SUBAPPLICATION Uebung_080e3 (* Beispiel für E_CTU mit Eventbremse durch E_D_FF_ANY *)
  (* Standard: 61499-2; Description: Copyright (c) 2023 Meisterschulen am Ostbahnhof This program and the accompanying materials are made available under the terms of the Eclipse Public License 2.0 which is available at https://www.eclipse.org/legal/epl-2.0/ SPDX-License-Identifier: EPL-2.0 *)
  (* Version 1.0, 2023-10-23, Franz Höpfinger, Meisterschulen am Ostbahnhof, initial API and implementation and/or initial documentation *)
  PACKAGE Uebungen;
  IMPORT logiBUS::io::DI::logiBUS_DI::Input_I1;
  IMPORT logiBUS::io::DI::logiBUS_DI::Input_I2;
  IMPORT logiBUS::io::DI::logiBUS_DI_Events::BUTTON_SINGLE_CLICK;
  IMPORT logiBUS::io::DQ::logiBUS_DO::Output_Q1;
  IMPORT Uebungen::const::UT::DefaultPool::OutputNumber_N1;
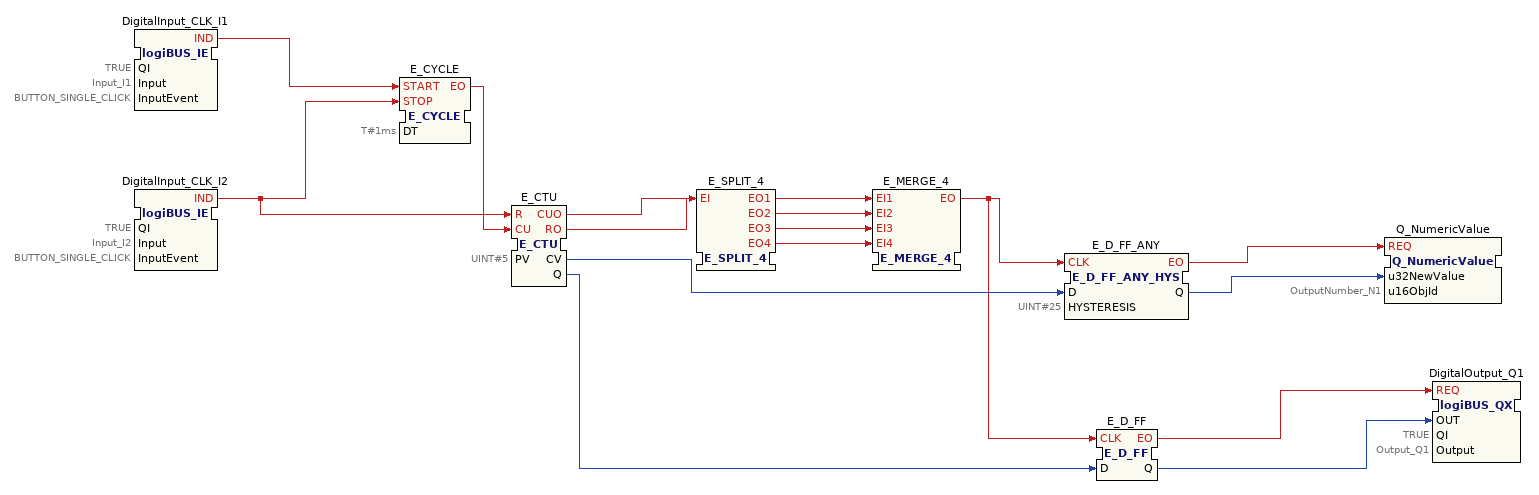
  FBS
    DigitalOutput_Q1 : logiBUS::io::DQ::logiBUS_QX(QI := TRUE, Output := Output_Q1);
    DigitalInput_CLK_I1 : logiBUS::io::DI::logiBUS_IE(QI := TRUE, Input := Input_I1, InputEvent := BUTTON_SINGLE_CLICK);
    E_CTU : iec61499::events::E_CTU(PV := UINT#5);
    DigitalInput_CLK_I2 : logiBUS::io::DI::logiBUS_IE(QI := TRUE, Input := Input_I2, InputEvent := BUTTON_SINGLE_CLICK);
    E_SPLIT_4 : iec61499::events::E_SPLIT_4;
    E_MERGE_4 : iec61499::events::E_MERGE_4;
    E_D_FF_ANY : logiBUS::signalprocessing::hysteresis::E_D_FF_ANY_HYS(HYSTERESIS := UINT#25);
    E_D_FF : iec61499::events::E_D_FF;
    Q_NumericValue : isobus::UT::Q::Q_NumericValue(u16ObjId := OutputNumber_N1);
    E_CYCLE : iec61499::events::E_CYCLE(DT := T#1ms);
  END_FBS
  EVENT_CONNECTIONS
    DigitalInput_CLK_I1.IND TO E_CYCLE.START;
    E_CTU.CUO TO E_SPLIT_4.EI;
    E_CTU.RO TO E_SPLIT_4.EI;
    DigitalInput_CLK_I2.IND TO E_CTU.R;
    E_SPLIT_4.EO1 TO E_MERGE_4.EI1;
    E_SPLIT_4.EO2 TO E_MERGE_4.EI2;
    E_SPLIT_4.EO3 TO E_MERGE_4.EI3;
    E_SPLIT_4.EO4 TO E_MERGE_4.EI4;
    E_MERGE_4.EO TO E_D_FF_ANY.CLK;
    E_D_FF_ANY.EO TO Q_NumericValue.REQ;
    E_MERGE_4.EO TO E_D_FF.CLK;
    E_D_FF.EO TO DigitalOutput_Q1.REQ;
    E_CYCLE.EO TO E_CTU.CU;
    DigitalInput_CLK_I2.IND TO E_CYCLE.STOP;
  END_CONNECTIONS
  DATA_CONNECTIONS
    E_CTU.CV TO E_D_FF_ANY.D;
    E_D_FF_ANY.Q TO Q_NumericValue.u32NewValue;
    E_CTU.Q TO E_D_FF.D;
    E_D_FF.Q TO DigitalOutput_Q1.OUT;
  END_CONNECTIONS
END_SUBAPPLICATION
